FUNCTION_BLOCK SimpleStateFeedbackController

VAR_INPUT
	xRobotPose: 		RobotPoseSimple; 				//current pose
	xRobotPoseRef: 		RobotPoseSimple; 				//reference pose
	xK:					ARRAY [0..2,0..2]  OF LREAL;  	//gain matrix K
END_VAR

VAR_OUTPUT
	//control outputs
	vXrobot:			LREAL;
	vYrobot:			LREAL;
	omegaRobot:			LREAL;
END_VAR

VAR
	poseError: RobotPoseSimple;
	u: ARRAY[0..2] OF LREAL;
	i: INT;
END_VAR

//1.) calculate pose errors
poseError.x 	:= xRobotPoseRef.x 		- xRobotPose.x;
poseError.y 	:= xRobotPoseRef.y 		- xRobotPose.y;
poseError.theta := xRobotPoseRef.theta 	- xRobotPose.theta;

//2.) apply gain on errors
FOR i := 0 TO 2 DO
	u[i] := xK[0,i] * poseError.x + xK[1,i] * poseError.y + xK[2,i] * poseError.theta;
END_FOR;

//3.) set control outputs
vXrobot 	:= u[0];
vYrobot 	:= u[1];
omegaRobot	:= u[2];

END_FUNCTION_BLOCK

(* stored: Version 1.1.0.1, ProductVersion 3.1.4024.11
   POU SimpleStateFeedbackController: Id {b6b00111-b334-4516-8a6e-fa6dcb5c765f}, SpecialFunc None *)
